Xinje XDPPro project, PLC1: XD5-60T10 (software 3.7.4b 2021-06-17)

PROGRAM Ladder

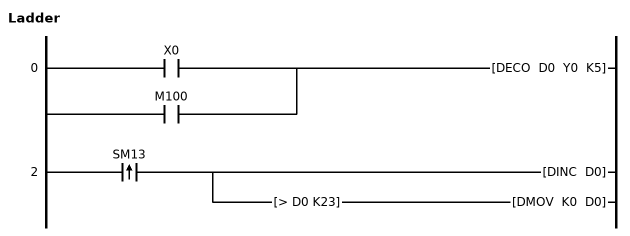
LD     X0
OR     M100
DECO   D0 Y0 K5
LDP    SM13
DINC   D0
AND>   D0 K23
DMOV   K0 D0